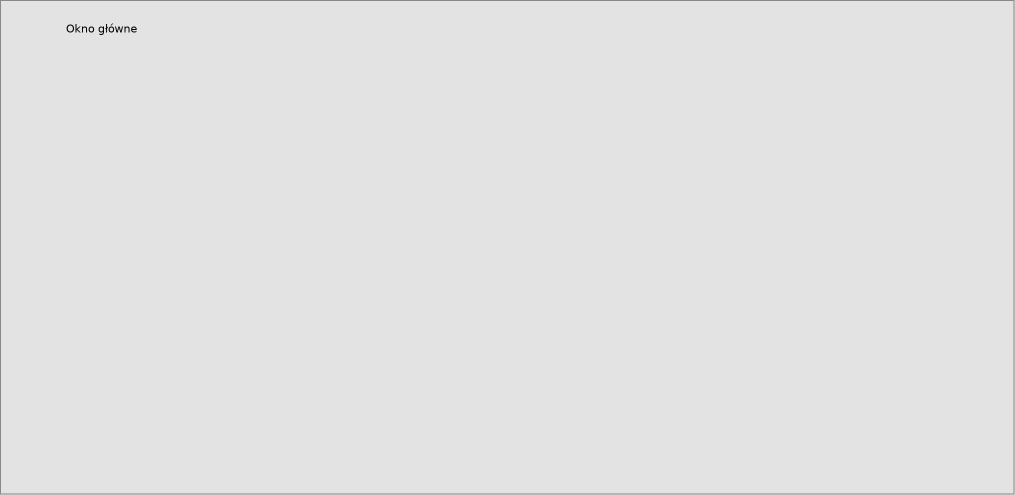
VISUALIZATION F_00_MainScreen  // 1015x495
    Label (27,14 150x30), "Okno główne"
END_VISUALIZATION

(* stored: Version 1.1.0.1
   Visu F_00_MainScreen: Id {72e12c18-5897-0561-10bd-c92fb2290c18} *)
